// Mitsubishi GX Works2 project: 正反转   PLC: FX1S

PROGRAM MAIN
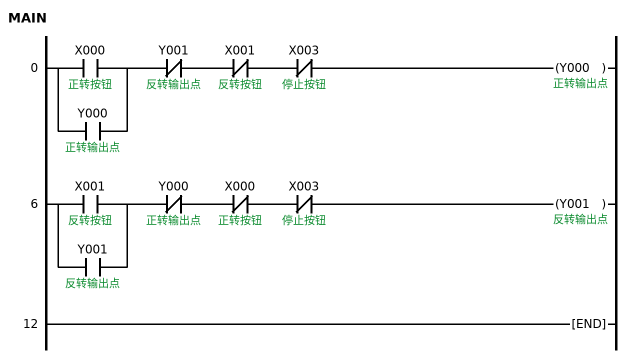
0     LD      X000  ; 正转按钮
      OR      Y000  ; 正转输出点
      ANI     Y001  ; 反转输出点
      ANI     X001  ; 反转按钮
      ANI     X003  ; 停止按钮
      OUT     Y000  ; 正转输出点
6     LD      X001  ; 反转按钮
      OR      Y001  ; 反转输出点
      ANI     Y000  ; 正转输出点
      ANI     X000  ; 正转按钮
      ANI     X003  ; 停止按钮
      OUT     Y001  ; 反转输出点
12    END
END_PROGRAM
